# EPICS substitutions: ek9000App/Db/EL4104.substitutions
file EL4104.template
{       pattern
        {
                TERMINAL,

        }
        {
        }
}
